// TIA Portal V20 export
FUNCTION "02 T5 EXCENTRIC HMI" : Void   // FC1218, LAD
TITLE = HMI
{ S7_Optimized_Access := 'TRUE' }
// stored: AutoNumber false, SetENOAutomatically false
BEGIN

REGION Network 1: Reset command interface from HMI in case of time-out
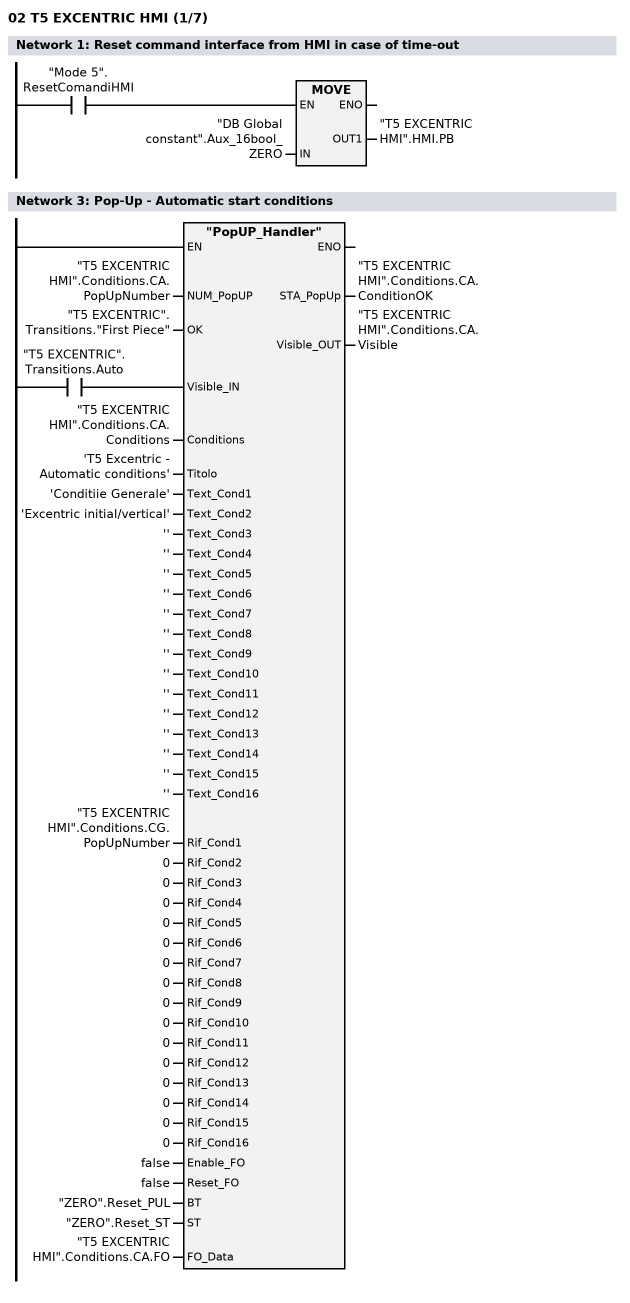
   RUNG wire#powerrail
      Contact( "Mode 5".ResetComandiHMI )
      Move(in := "DB Global constant".Aux_16bool_ZERO, out1 => "T5 EXCENTRIC HMI".HMI.PB)
   END_RUNG
   // the same network as SCL:
   IF "Mode 5".ResetComandiHMI THEN
       "T5 EXCENTRIC HMI".HMI.PB := "DB Global constant".Aux_16bool_ZERO;
   END_IF;
END_REGION

REGION Network 2: ============ POP UP ============
END_REGION

REGION Network 3: Pop-Up - Automatic start conditions
   RUNG wire#powerrail
      "PopUP_Handler"(Visible_IN := wire#w1, NUM_PopUP := "T5 EXCENTRIC HMI".Conditions.CA.PopUpNumber, OK := "T5 EXCENTRIC".Transitions."First Piece", Conditions := "T5 EXCENTRIC HMI".Conditions.CA.Conditions, Titolo := 'T5 Excentric - Automatic conditions', Text_Cond1 := 'Conditiie Generale', Text_Cond2 := 'Excentric initial/vertical', Text_Cond3 := '', Text_Cond4 := '', Text_Cond5 := '', Text_Cond6 := '', Text_Cond7 := '', Text_Cond8 := '', Text_Cond9 := '', Text_Cond10 := '', Text_Cond11 := '', Text_Cond12 := '', Text_Cond13 := '', Text_Cond14 := '', Text_Cond15 := '', Text_Cond16 := '', Rif_Cond1 := "T5 EXCENTRIC HMI".Conditions.CG.PopUpNumber, Rif_Cond2 := 0, Rif_Cond3 := 0, Rif_Cond4 := 0, Rif_Cond5 := 0, Rif_Cond6 := 0, Rif_Cond7 := 0, Rif_Cond8 := 0, Rif_Cond9 := 0, Rif_Cond10 := 0, Rif_Cond11 := 0, Rif_Cond12 := 0, Rif_Cond13 := 0, Rif_Cond14 := 0, Rif_Cond15 := 0, Rif_Cond16 := 0, Enable_FO := false, Reset_FO := false, BT := "ZERO".Reset_PUL, ST := "ZERO".Reset_ST, FO_Data := "T5 EXCENTRIC HMI".Conditions.CA.FO, STA_PopUp => "T5 EXCENTRIC HMI".Conditions.CA.ConditionOK, Visible_OUT => "T5 EXCENTRIC HMI".Conditions.CA.Visible)
   END_RUNG
   RUNG wire#powerrail
      Contact( "T5 EXCENTRIC".Transitions.Auto )
   END_RUNG wire#w1
   // the same network as SCL:
   "PopUP_Handler"(NUM_PopUP := "T5 EXCENTRIC HMI".Conditions.CA.PopUpNumber,
                   OK := "T5 EXCENTRIC".Transitions."First Piece",
                   Visible_IN := "T5 EXCENTRIC".Transitions.Auto,
                   Conditions := "T5 EXCENTRIC HMI".Conditions.CA.Conditions,
                   Titolo := 'T5 Excentric - Automatic conditions',
                   Text_Cond1 := 'Conditiie Generale',
                   Text_Cond2 := 'Excentric initial/vertical',
                   Text_Cond3 := '',
                   Text_Cond4 := '',
                   Text_Cond5 := '',
                   Text_Cond6 := '',
                   Text_Cond7 := '',
                   Text_Cond8 := '',
                   Text_Cond9 := '',
                   Text_Cond10 := '',
                   Text_Cond11 := '',
                   Text_Cond12 := '',
                   Text_Cond13 := '',
                   Text_Cond14 := '',
                   Text_Cond15 := '',
                   Text_Cond16 := '',
                   Rif_Cond1 := "T5 EXCENTRIC HMI".Conditions.CG.PopUpNumber,
                   Rif_Cond2 := 0,
                   Rif_Cond3 := 0,
                   Rif_Cond4 := 0,
                   Rif_Cond5 := 0,
                   Rif_Cond6 := 0,
                   Rif_Cond7 := 0,
                   Rif_Cond8 := 0,
                   Rif_Cond9 := 0,
                   Rif_Cond10 := 0,
                   Rif_Cond11 := 0,
                   Rif_Cond12 := 0,
                   Rif_Cond13 := 0,
                   Rif_Cond14 := 0,
                   Rif_Cond15 := 0,
                   Rif_Cond16 := 0,
                   Enable_FO := false,
                   Reset_FO := false,
                   BT := "ZERO".Reset_PUL,
                   ST := "ZERO".Reset_ST,
                   FO_Data := "T5 EXCENTRIC HMI".Conditions.CA.FO,
                   STA_PopUp => "T5 EXCENTRIC HMI".Conditions.CA.ConditionOK,
                   Visible_OUT => "T5 EXCENTRIC HMI".Conditions.CA.Visible);
END_REGION

REGION Network 4: Pop-Up - General conditions
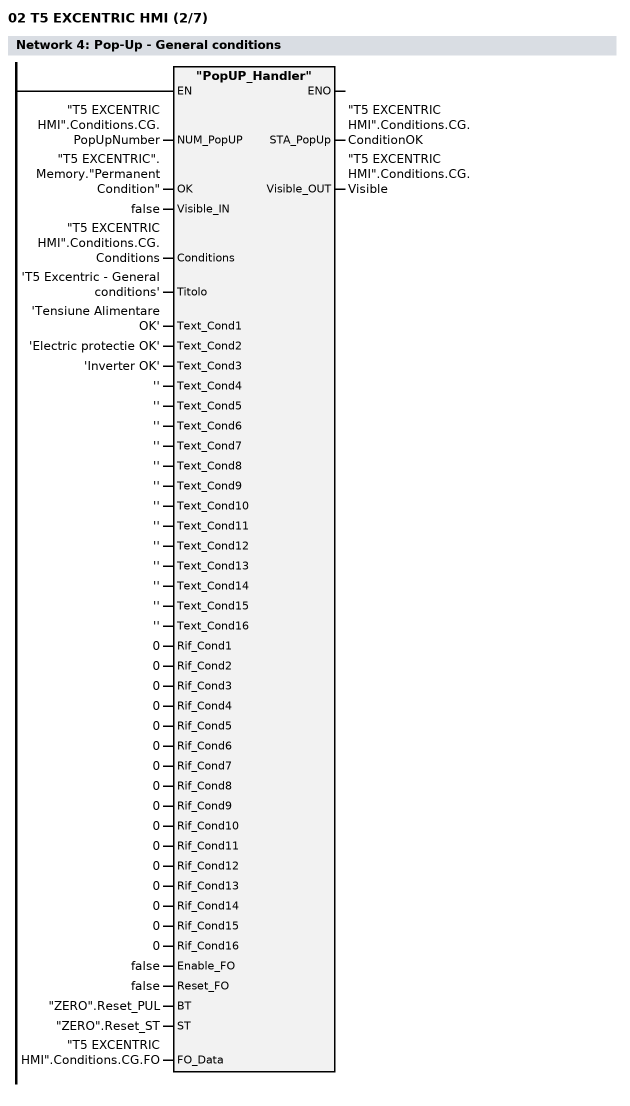
   RUNG wire#powerrail
      "PopUP_Handler"(NUM_PopUP := "T5 EXCENTRIC HMI".Conditions.CG.PopUpNumber, OK := "T5 EXCENTRIC".Memory."Permanent Condition", Visible_IN := false, Conditions := "T5 EXCENTRIC HMI".Conditions.CG.Conditions, Titolo := 'T5 Excentric - General conditions', Text_Cond1 := 'Tensiune Alimentare OK', Text_Cond2 := 'Electric protectie OK', Text_Cond3 := 'Inverter OK', Text_Cond4 := '', Text_Cond5 := '', Text_Cond6 := '', Text_Cond7 := '', Text_Cond8 := '', Text_Cond9 := '', Text_Cond10 := '', Text_Cond11 := '', Text_Cond12 := '', Text_Cond13 := '', Text_Cond14 := '', Text_Cond15 := '', Text_Cond16 := '', Rif_Cond1 := 0, Rif_Cond2 := 0, Rif_Cond3 := 0, Rif_Cond4 := 0, Rif_Cond5 := 0, Rif_Cond6 := 0, Rif_Cond7 := 0, Rif_Cond8 := 0, Rif_Cond9 := 0, Rif_Cond10 := 0, Rif_Cond11 := 0, Rif_Cond12 := 0, Rif_Cond13 := 0, Rif_Cond14 := 0, Rif_Cond15 := 0, Rif_Cond16 := 0, Enable_FO := false, Reset_FO := false, BT := "ZERO".Reset_PUL, ST := "ZERO".Reset_ST, FO_Data := "T5 EXCENTRIC HMI".Conditions.CG.FO, STA_PopUp => "T5 EXCENTRIC HMI".Conditions.CG.ConditionOK, Visible_OUT => "T5 EXCENTRIC HMI".Conditions.CG.Visible)
   END_RUNG
   // the same network as SCL:
   "PopUP_Handler"(NUM_PopUP := "T5 EXCENTRIC HMI".Conditions.CG.PopUpNumber,
                   OK := "T5 EXCENTRIC".Memory."Permanent Condition",
                   Visible_IN := false,
                   Conditions := "T5 EXCENTRIC HMI".Conditions.CG.Conditions,
                   Titolo := 'T5 Excentric - General conditions',
                   Text_Cond1 := 'Tensiune Alimentare OK',
                   Text_Cond2 := 'Electric protectie OK',
                   Text_Cond3 := 'Inverter OK',
                   Text_Cond4 := '',
                   Text_Cond5 := '',
                   Text_Cond6 := '',
                   Text_Cond7 := '',
                   Text_Cond8 := '',
                   Text_Cond9 := '',
                   Text_Cond10 := '',
                   Text_Cond11 := '',
                   Text_Cond12 := '',
                   Text_Cond13 := '',
                   Text_Cond14 := '',
                   Text_Cond15 := '',
                   Text_Cond16 := '',
                   Rif_Cond1 := 0,
                   Rif_Cond2 := 0,
                   Rif_Cond3 := 0,
                   Rif_Cond4 := 0,
                   Rif_Cond5 := 0,
                   Rif_Cond6 := 0,
                   Rif_Cond7 := 0,
                   Rif_Cond8 := 0,
                   Rif_Cond9 := 0,
                   Rif_Cond10 := 0,
                   Rif_Cond11 := 0,
                   Rif_Cond12 := 0,
                   Rif_Cond13 := 0,
                   Rif_Cond14 := 0,
                   Rif_Cond15 := 0,
                   Rif_Cond16 := 0,
                   Enable_FO := false,
                   Reset_FO := false,
                   BT := "ZERO".Reset_PUL,
                   ST := "ZERO".Reset_ST,
                   FO_Data := "T5 EXCENTRIC HMI".Conditions.CG.FO,
                   STA_PopUp => "T5 EXCENTRIC HMI".Conditions.CG.ConditionOK,
                   Visible_OUT => "T5 EXCENTRIC HMI".Conditions.CG.Visible);
END_REGION

REGION Network 5: Pop-Up - Cycle start conditions - Initial
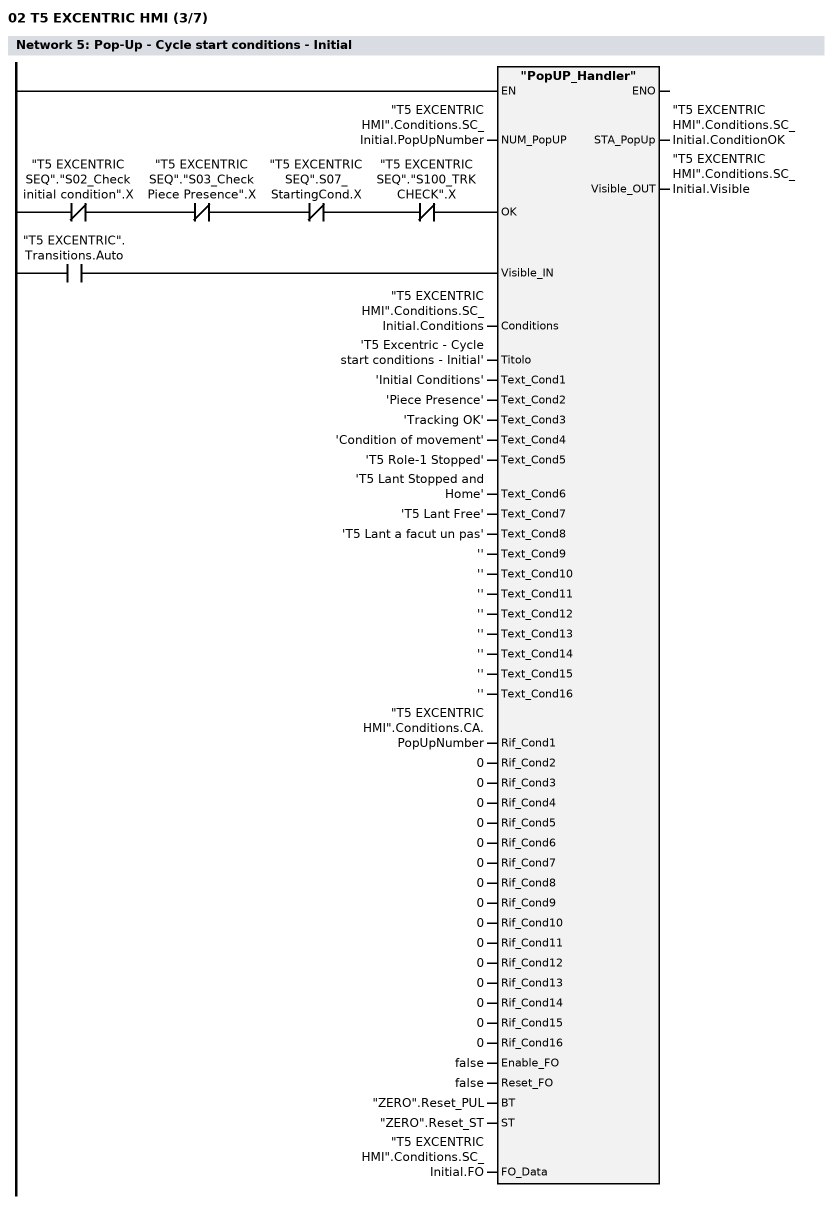
   RUNG wire#powerrail
      "PopUP_Handler"(OK := wire#w1, Visible_IN := wire#w2, NUM_PopUP := "T5 EXCENTRIC HMI".Conditions.SC_Initial.PopUpNumber, Conditions := "T5 EXCENTRIC HMI".Conditions.SC_Initial.Conditions, Titolo := 'T5 Excentric - Cycle start conditions - Initial', Text_Cond1 := 'Initial Conditions', Text_Cond2 := 'Piece Presence', Text_Cond3 := 'Tracking OK', Text_Cond4 := 'Condition of movement', Text_Cond5 := 'T5 Role-1 Stopped', Text_Cond6 := 'T5 Lant Stopped and Home', Text_Cond7 := 'T5 Lant Free', Text_Cond8 := 'T5 Lant a facut un pas', Text_Cond9 := '', Text_Cond10 := '', Text_Cond11 := '', Text_Cond12 := '', Text_Cond13 := '', Text_Cond14 := '', Text_Cond15 := '', Text_Cond16 := '', Rif_Cond1 := "T5 EXCENTRIC HMI".Conditions.CA.PopUpNumber, Rif_Cond2 := 0, Rif_Cond3 := 0, Rif_Cond4 := 0, Rif_Cond5 := 0, Rif_Cond6 := 0, Rif_Cond7 := 0, Rif_Cond8 := 0, Rif_Cond9 := 0, Rif_Cond10 := 0, Rif_Cond11 := 0, Rif_Cond12 := 0, Rif_Cond13 := 0, Rif_Cond14 := 0, Rif_Cond15 := 0, Rif_Cond16 := 0, Enable_FO := false, Reset_FO := false, BT := "ZERO".Reset_PUL, ST := "ZERO".Reset_ST, FO_Data := "T5 EXCENTRIC HMI".Conditions.SC_Initial.FO, STA_PopUp => "T5 EXCENTRIC HMI".Conditions.SC_Initial.ConditionOK, Visible_OUT => "T5 EXCENTRIC HMI".Conditions.SC_Initial.Visible)
   END_RUNG
   RUNG wire#powerrail
      I_Contact( "T5 EXCENTRIC SEQ"."S02_Check initial condition".X )
      I_Contact( "T5 EXCENTRIC SEQ"."S03_Check Piece Presence".X )
      I_Contact( "T5 EXCENTRIC SEQ".S07_StartingCond.X )
      I_Contact( "T5 EXCENTRIC SEQ"."S100_TRK CHECK".X )
   END_RUNG wire#w1
   RUNG wire#powerrail
      Contact( "T5 EXCENTRIC".Transitions.Auto )
   END_RUNG wire#w2
   // the same network as SCL:
   "PopUP_Handler"(NUM_PopUP := "T5 EXCENTRIC HMI".Conditions.SC_Initial.PopUpNumber,
                   OK := NOT "T5 EXCENTRIC SEQ"."S02_Check initial condition".X AND NOT "T5 EXCENTRIC SEQ"."S03_Check Piece Presence".X AND NOT "T5 EXCENTRIC SEQ".S07_StartingCond.X AND NOT "T5 EXCENTRIC SEQ"."S100_TRK CHECK".X,
                   Visible_IN := "T5 EXCENTRIC".Transitions.Auto,
                   Conditions := "T5 EXCENTRIC HMI".Conditions.SC_Initial.Conditions,
                   Titolo := 'T5 Excentric - Cycle start conditions - Initial',
                   Text_Cond1 := 'Initial Conditions',
                   Text_Cond2 := 'Piece Presence',
                   Text_Cond3 := 'Tracking OK',
                   Text_Cond4 := 'Condition of movement',
                   Text_Cond5 := 'T5 Role-1 Stopped',
                   Text_Cond6 := 'T5 Lant Stopped and Home',
                   Text_Cond7 := 'T5 Lant Free',
                   Text_Cond8 := 'T5 Lant a facut un pas',
                   Text_Cond9 := '',
                   Text_Cond10 := '',
                   Text_Cond11 := '',
                   Text_Cond12 := '',
                   Text_Cond13 := '',
                   Text_Cond14 := '',
                   Text_Cond15 := '',
                   Text_Cond16 := '',
                   Rif_Cond1 := "T5 EXCENTRIC HMI".Conditions.CA.PopUpNumber,
                   Rif_Cond2 := 0,
                   Rif_Cond3 := 0,
                   Rif_Cond4 := 0,
                   Rif_Cond5 := 0,
                   Rif_Cond6 := 0,
                   Rif_Cond7 := 0,
                   Rif_Cond8 := 0,
                   Rif_Cond9 := 0,
                   Rif_Cond10 := 0,
                   Rif_Cond11 := 0,
                   Rif_Cond12 := 0,
                   Rif_Cond13 := 0,
                   Rif_Cond14 := 0,
                   Rif_Cond15 := 0,
                   Rif_Cond16 := 0,
                   Enable_FO := false,
                   Reset_FO := false,
                   BT := "ZERO".Reset_PUL,
                   ST := "ZERO".Reset_ST,
                   FO_Data := "T5 EXCENTRIC HMI".Conditions.SC_Initial.FO,
                   STA_PopUp => "T5 EXCENTRIC HMI".Conditions.SC_Initial.ConditionOK,
                   Visible_OUT => "T5 EXCENTRIC HMI".Conditions.SC_Initial.Visible);
END_REGION

REGION Network 6: Pop-Up - Cycle start conditions - Vertical
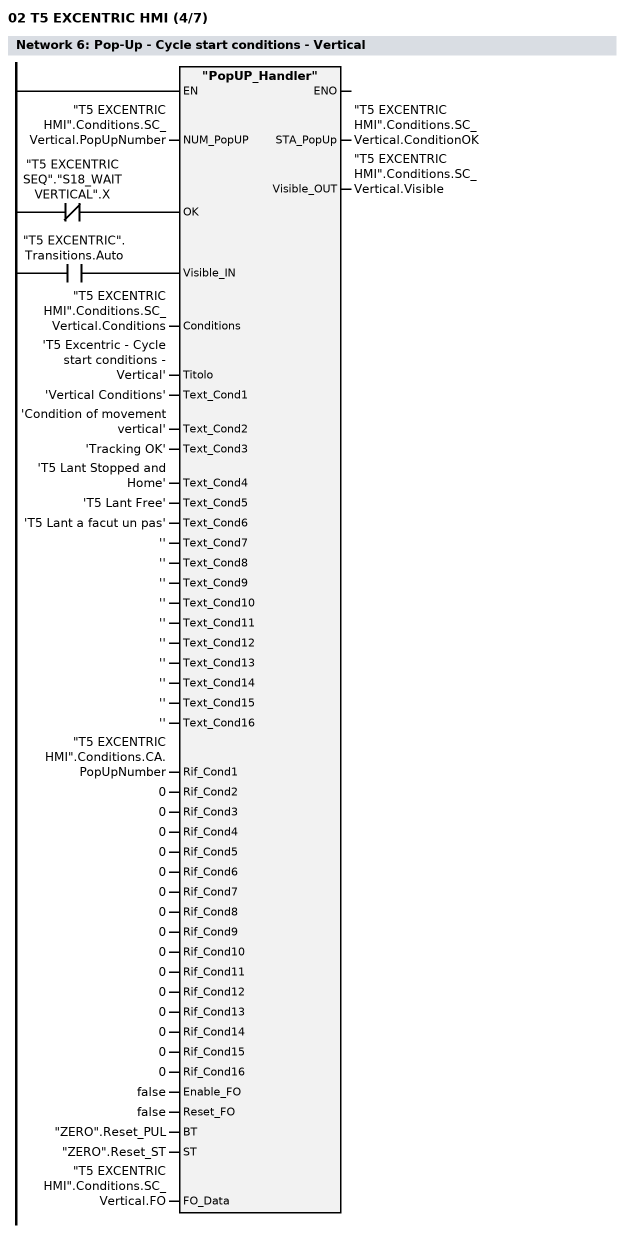
   RUNG wire#powerrail
      "PopUP_Handler"(OK := wire#w1, Visible_IN := wire#w2, NUM_PopUP := "T5 EXCENTRIC HMI".Conditions.SC_Vertical.PopUpNumber, Conditions := "T5 EXCENTRIC HMI".Conditions.SC_Vertical.Conditions, Titolo := 'T5 Excentric - Cycle start conditions - Vertical', Text_Cond1 := 'Vertical Conditions', Text_Cond2 := 'Condition of movement vertical', Text_Cond3 := 'Tracking OK', Text_Cond4 := 'T5 Lant Stopped and Home', Text_Cond5 := 'T5 Lant Free', Text_Cond6 := 'T5 Lant a facut un pas', Text_Cond7 := '', Text_Cond8 := '', Text_Cond9 := '', Text_Cond10 := '', Text_Cond11 := '', Text_Cond12 := '', Text_Cond13 := '', Text_Cond14 := '', Text_Cond15 := '', Text_Cond16 := '', Rif_Cond1 := "T5 EXCENTRIC HMI".Conditions.CA.PopUpNumber, Rif_Cond2 := 0, Rif_Cond3 := 0, Rif_Cond4 := 0, Rif_Cond5 := 0, Rif_Cond6 := 0, Rif_Cond7 := 0, Rif_Cond8 := 0, Rif_Cond9 := 0, Rif_Cond10 := 0, Rif_Cond11 := 0, Rif_Cond12 := 0, Rif_Cond13 := 0, Rif_Cond14 := 0, Rif_Cond15 := 0, Rif_Cond16 := 0, Enable_FO := false, Reset_FO := false, BT := "ZERO".Reset_PUL, ST := "ZERO".Reset_ST, FO_Data := "T5 EXCENTRIC HMI".Conditions.SC_Vertical.FO, STA_PopUp => "T5 EXCENTRIC HMI".Conditions.SC_Vertical.ConditionOK, Visible_OUT => "T5 EXCENTRIC HMI".Conditions.SC_Vertical.Visible)
   END_RUNG
   RUNG wire#powerrail
      I_Contact( "T5 EXCENTRIC SEQ"."S18_WAIT VERTICAL".X )
   END_RUNG wire#w1
   RUNG wire#powerrail
      Contact( "T5 EXCENTRIC".Transitions.Auto )
   END_RUNG wire#w2
   // the same network as SCL:
   "PopUP_Handler"(NUM_PopUP := "T5 EXCENTRIC HMI".Conditions.SC_Vertical.PopUpNumber,
                   OK := NOT "T5 EXCENTRIC SEQ"."S18_WAIT VERTICAL".X,
                   Visible_IN := "T5 EXCENTRIC".Transitions.Auto,
                   Conditions := "T5 EXCENTRIC HMI".Conditions.SC_Vertical.Conditions,
                   Titolo := 'T5 Excentric - Cycle start conditions - Vertical',
                   Text_Cond1 := 'Vertical Conditions',
                   Text_Cond2 := 'Condition of movement vertical',
                   Text_Cond3 := 'Tracking OK',
                   Text_Cond4 := 'T5 Lant Stopped and Home',
                   Text_Cond5 := 'T5 Lant Free',
                   Text_Cond6 := 'T5 Lant a facut un pas',
                   Text_Cond7 := '',
                   Text_Cond8 := '',
                   Text_Cond9 := '',
                   Text_Cond10 := '',
                   Text_Cond11 := '',
                   Text_Cond12 := '',
                   Text_Cond13 := '',
                   Text_Cond14 := '',
                   Text_Cond15 := '',
                   Text_Cond16 := '',
                   Rif_Cond1 := "T5 EXCENTRIC HMI".Conditions.CA.PopUpNumber,
                   Rif_Cond2 := 0,
                   Rif_Cond3 := 0,
                   Rif_Cond4 := 0,
                   Rif_Cond5 := 0,
                   Rif_Cond6 := 0,
                   Rif_Cond7 := 0,
                   Rif_Cond8 := 0,
                   Rif_Cond9 := 0,
                   Rif_Cond10 := 0,
                   Rif_Cond11 := 0,
                   Rif_Cond12 := 0,
                   Rif_Cond13 := 0,
                   Rif_Cond14 := 0,
                   Rif_Cond15 := 0,
                   Rif_Cond16 := 0,
                   Enable_FO := false,
                   Reset_FO := false,
                   BT := "ZERO".Reset_PUL,
                   ST := "ZERO".Reset_ST,
                   FO_Data := "T5 EXCENTRIC HMI".Conditions.SC_Vertical.FO,
                   STA_PopUp => "T5 EXCENTRIC HMI".Conditions.SC_Vertical.ConditionOK,
                   Visible_OUT => "T5 EXCENTRIC HMI".Conditions.SC_Vertical.Visible);
END_REGION

REGION Network 7: Pop-Up - Conditions of movement FORWARD
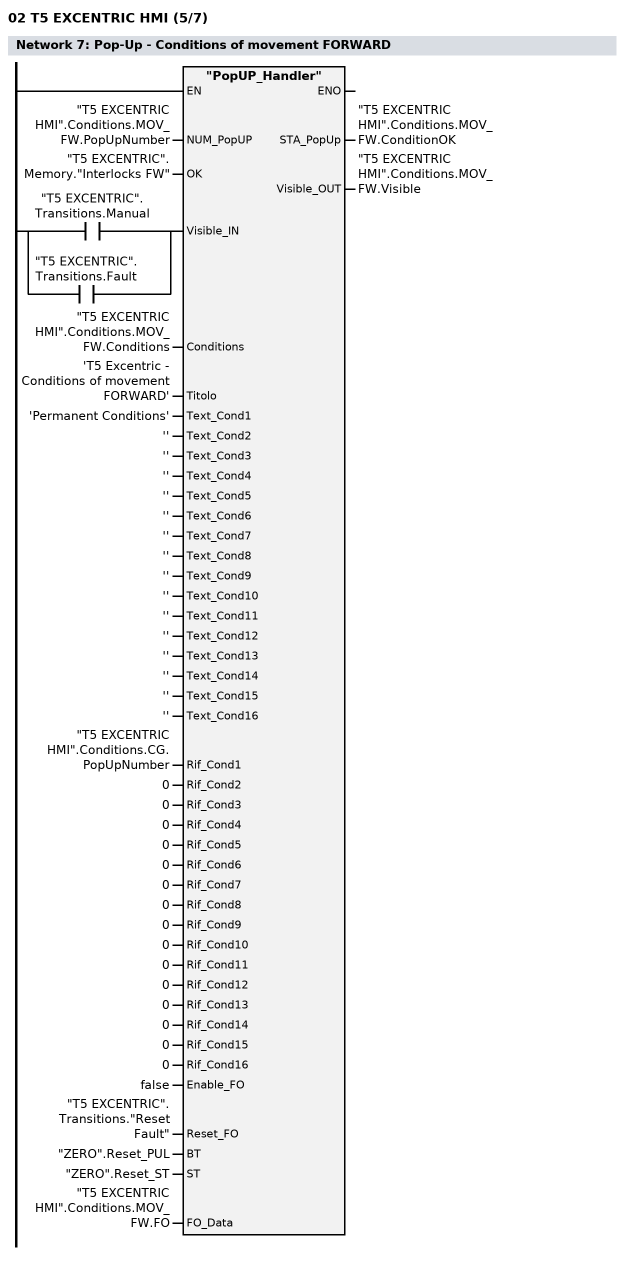
   RUNG wire#powerrail
      "PopUP_Handler"(Visible_IN := wire#w1, NUM_PopUP := "T5 EXCENTRIC HMI".Conditions.MOV_FW.PopUpNumber, OK := "T5 EXCENTRIC".Memory."Interlocks FW", Conditions := "T5 EXCENTRIC HMI".Conditions.MOV_FW.Conditions, Titolo := 'T5 Excentric - Conditions of movement FORWARD', Text_Cond1 := 'Permanent Conditions', Text_Cond2 := '', Text_Cond3 := '', Text_Cond4 := '', Text_Cond5 := '', Text_Cond6 := '', Text_Cond7 := '', Text_Cond8 := '', Text_Cond9 := '', Text_Cond10 := '', Text_Cond11 := '', Text_Cond12 := '', Text_Cond13 := '', Text_Cond14 := '', Text_Cond15 := '', Text_Cond16 := '', Rif_Cond1 := "T5 EXCENTRIC HMI".Conditions.CG.PopUpNumber, Rif_Cond2 := 0, Rif_Cond3 := 0, Rif_Cond4 := 0, Rif_Cond5 := 0, Rif_Cond6 := 0, Rif_Cond7 := 0, Rif_Cond8 := 0, Rif_Cond9 := 0, Rif_Cond10 := 0, Rif_Cond11 := 0, Rif_Cond12 := 0, Rif_Cond13 := 0, Rif_Cond14 := 0, Rif_Cond15 := 0, Rif_Cond16 := 0, Enable_FO := false, Reset_FO := "T5 EXCENTRIC".Transitions."Reset Fault", BT := "ZERO".Reset_PUL, ST := "ZERO".Reset_ST, FO_Data := "T5 EXCENTRIC HMI".Conditions.MOV_FW.FO, STA_PopUp => "T5 EXCENTRIC HMI".Conditions.MOV_FW.ConditionOK, Visible_OUT => "T5 EXCENTRIC HMI".Conditions.MOV_FW.Visible)
   END_RUNG
   RUNG wire#powerrail
      Contact( "T5 EXCENTRIC".Transitions.Manual )
   END_RUNG wire#w1
   RUNG wire#powerrail
      Contact( "T5 EXCENTRIC".Transitions.Fault )
   END_RUNG wire#w1
   // the same network as SCL:
   "PopUP_Handler"(NUM_PopUP := "T5 EXCENTRIC HMI".Conditions.MOV_FW.PopUpNumber,
                   OK := "T5 EXCENTRIC".Memory."Interlocks FW",
                   Visible_IN := "T5 EXCENTRIC".Transitions.Manual OR "T5 EXCENTRIC".Transitions.Fault,
                   Conditions := "T5 EXCENTRIC HMI".Conditions.MOV_FW.Conditions,
                   Titolo := 'T5 Excentric - Conditions of movement FORWARD',
                   Text_Cond1 := 'Permanent Conditions',
                   Text_Cond2 := '',
                   Text_Cond3 := '',
                   Text_Cond4 := '',
                   Text_Cond5 := '',
                   Text_Cond6 := '',
                   Text_Cond7 := '',
                   Text_Cond8 := '',
                   Text_Cond9 := '',
                   Text_Cond10 := '',
                   Text_Cond11 := '',
                   Text_Cond12 := '',
                   Text_Cond13 := '',
                   Text_Cond14 := '',
                   Text_Cond15 := '',
                   Text_Cond16 := '',
                   Rif_Cond1 := "T5 EXCENTRIC HMI".Conditions.CG.PopUpNumber,
                   Rif_Cond2 := 0,
                   Rif_Cond3 := 0,
                   Rif_Cond4 := 0,
                   Rif_Cond5 := 0,
                   Rif_Cond6 := 0,
                   Rif_Cond7 := 0,
                   Rif_Cond8 := 0,
                   Rif_Cond9 := 0,
                   Rif_Cond10 := 0,
                   Rif_Cond11 := 0,
                   Rif_Cond12 := 0,
                   Rif_Cond13 := 0,
                   Rif_Cond14 := 0,
                   Rif_Cond15 := 0,
                   Rif_Cond16 := 0,
                   Enable_FO := false,
                   Reset_FO := "T5 EXCENTRIC".Transitions."Reset Fault",
                   BT := "ZERO".Reset_PUL,
                   ST := "ZERO".Reset_ST,
                   FO_Data := "T5 EXCENTRIC HMI".Conditions.MOV_FW.FO,
                   STA_PopUp => "T5 EXCENTRIC HMI".Conditions.MOV_FW.ConditionOK,
                   Visible_OUT => "T5 EXCENTRIC HMI".Conditions.MOV_FW.Visible);
END_REGION

REGION Network 8: Pop-Up - Conditions of movement BACKWARD
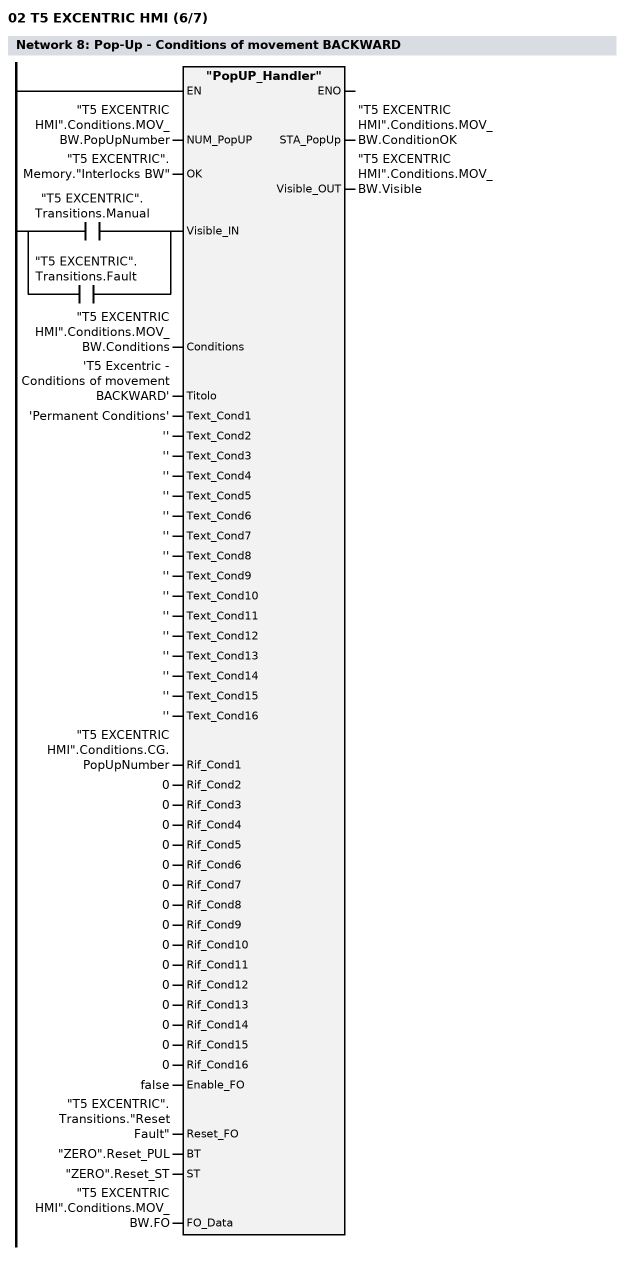
   RUNG wire#powerrail
      "PopUP_Handler"(Visible_IN := wire#w1, NUM_PopUP := "T5 EXCENTRIC HMI".Conditions.MOV_BW.PopUpNumber, OK := "T5 EXCENTRIC".Memory."Interlocks BW", Conditions := "T5 EXCENTRIC HMI".Conditions.MOV_BW.Conditions, Titolo := 'T5 Excentric - Conditions of movement BACKWARD', Text_Cond1 := 'Permanent Conditions', Text_Cond2 := '', Text_Cond3 := '', Text_Cond4 := '', Text_Cond5 := '', Text_Cond6 := '', Text_Cond7 := '', Text_Cond8 := '', Text_Cond9 := '', Text_Cond10 := '', Text_Cond11 := '', Text_Cond12 := '', Text_Cond13 := '', Text_Cond14 := '', Text_Cond15 := '', Text_Cond16 := '', Rif_Cond1 := "T5 EXCENTRIC HMI".Conditions.CG.PopUpNumber, Rif_Cond2 := 0, Rif_Cond3 := 0, Rif_Cond4 := 0, Rif_Cond5 := 0, Rif_Cond6 := 0, Rif_Cond7 := 0, Rif_Cond8 := 0, Rif_Cond9 := 0, Rif_Cond10 := 0, Rif_Cond11 := 0, Rif_Cond12 := 0, Rif_Cond13 := 0, Rif_Cond14 := 0, Rif_Cond15 := 0, Rif_Cond16 := 0, Enable_FO := false, Reset_FO := "T5 EXCENTRIC".Transitions."Reset Fault", BT := "ZERO".Reset_PUL, ST := "ZERO".Reset_ST, FO_Data := "T5 EXCENTRIC HMI".Conditions.MOV_BW.FO, STA_PopUp => "T5 EXCENTRIC HMI".Conditions.MOV_BW.ConditionOK, Visible_OUT => "T5 EXCENTRIC HMI".Conditions.MOV_BW.Visible)
   END_RUNG
   RUNG wire#powerrail
      Contact( "T5 EXCENTRIC".Transitions.Manual )
   END_RUNG wire#w1
   RUNG wire#powerrail
      Contact( "T5 EXCENTRIC".Transitions.Fault )
   END_RUNG wire#w1
   // the same network as SCL:
   "PopUP_Handler"(NUM_PopUP := "T5 EXCENTRIC HMI".Conditions.MOV_BW.PopUpNumber,
                   OK := "T5 EXCENTRIC".Memory."Interlocks BW",
                   Visible_IN := "T5 EXCENTRIC".Transitions.Manual OR "T5 EXCENTRIC".Transitions.Fault,
                   Conditions := "T5 EXCENTRIC HMI".Conditions.MOV_BW.Conditions,
                   Titolo := 'T5 Excentric - Conditions of movement BACKWARD',
                   Text_Cond1 := 'Permanent Conditions',
                   Text_Cond2 := '',
                   Text_Cond3 := '',
                   Text_Cond4 := '',
                   Text_Cond5 := '',
                   Text_Cond6 := '',
                   Text_Cond7 := '',
                   Text_Cond8 := '',
                   Text_Cond9 := '',
                   Text_Cond10 := '',
                   Text_Cond11 := '',
                   Text_Cond12 := '',
                   Text_Cond13 := '',
                   Text_Cond14 := '',
                   Text_Cond15 := '',
                   Text_Cond16 := '',
                   Rif_Cond1 := "T5 EXCENTRIC HMI".Conditions.CG.PopUpNumber,
                   Rif_Cond2 := 0,
                   Rif_Cond3 := 0,
                   Rif_Cond4 := 0,
                   Rif_Cond5 := 0,
                   Rif_Cond6 := 0,
                   Rif_Cond7 := 0,
                   Rif_Cond8 := 0,
                   Rif_Cond9 := 0,
                   Rif_Cond10 := 0,
                   Rif_Cond11 := 0,
                   Rif_Cond12 := 0,
                   Rif_Cond13 := 0,
                   Rif_Cond14 := 0,
                   Rif_Cond15 := 0,
                   Rif_Cond16 := 0,
                   Enable_FO := false,
                   Reset_FO := "T5 EXCENTRIC".Transitions."Reset Fault",
                   BT := "ZERO".Reset_PUL,
                   ST := "ZERO".Reset_ST,
                   FO_Data := "T5 EXCENTRIC HMI".Conditions.MOV_BW.FO,
                   STA_PopUp => "T5 EXCENTRIC HMI".Conditions.MOV_BW.ConditionOK,
                   Visible_OUT => "T5 EXCENTRIC HMI".Conditions.MOV_BW.Visible);
END_REGION

REGION Network 9: ============ HMI STATE ============
END_REGION

REGION Network 10: HMI Status - Commands
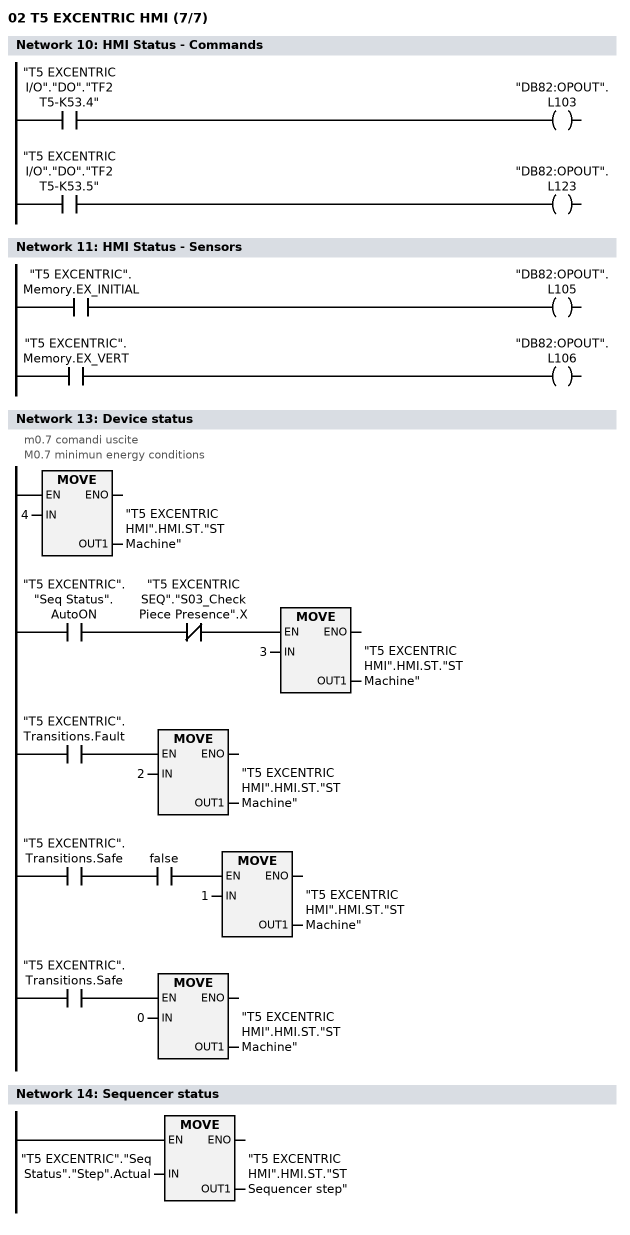
   RUNG wire#powerrail
      Contact( "T5 EXCENTRIC I/O"."DO"."TF2 T5-K53.4" )
      Coil( "DB82:OPOUT".L103 )
   END_RUNG
   RUNG wire#powerrail
      Contact( "T5 EXCENTRIC I/O"."DO"."TF2 T5-K53.5" )
      Coil( "DB82:OPOUT".L123 )
   END_RUNG
   // the same network as SCL:
   "DB82:OPOUT".L103 := "T5 EXCENTRIC I/O"."DO"."TF2 T5-K53.4";
   "DB82:OPOUT".L123 := "T5 EXCENTRIC I/O"."DO"."TF2 T5-K53.5";
END_REGION

REGION Network 11: HMI Status - Sensors
   RUNG wire#powerrail
      Contact( "T5 EXCENTRIC".Memory.EX_INITIAL )
      Coil( "DB82:OPOUT".L105 )
   END_RUNG
   RUNG wire#powerrail
      Contact( "T5 EXCENTRIC".Memory.EX_VERT )
      Coil( "DB82:OPOUT".L106 )
   END_RUNG
   // the same network as SCL:
   "DB82:OPOUT".L105 := "T5 EXCENTRIC".Memory.EX_INITIAL;
   "DB82:OPOUT".L106 := "T5 EXCENTRIC".Memory.EX_VERT;
END_REGION

REGION Network 12: HMI Status - Alarma
END_REGION

REGION Network 13: Device status
   // m0.7 comandi uscite
   // M0.7 minimun energy conditions
   RUNG wire#powerrail
      Move(in := 4, out1 => "T5 EXCENTRIC HMI".HMI.ST."ST Machine")
   END_RUNG
   RUNG wire#powerrail
      Contact( "T5 EXCENTRIC"."Seq Status".AutoON )
      I_Contact( "T5 EXCENTRIC SEQ"."S03_Check Piece Presence".X )
      Move(in := 3, out1 => "T5 EXCENTRIC HMI".HMI.ST."ST Machine")
   END_RUNG
   RUNG wire#powerrail
      Contact( "T5 EXCENTRIC".Transitions.Fault )
      Move(in := 2, out1 => "T5 EXCENTRIC HMI".HMI.ST."ST Machine")
   END_RUNG
   RUNG wire#powerrail
      Contact( "T5 EXCENTRIC".Transitions.Safe )
      Contact( false )
      Move(in := 1, out1 => "T5 EXCENTRIC HMI".HMI.ST."ST Machine")
   END_RUNG
   RUNG wire#powerrail
      Contact( "T5 EXCENTRIC".Transitions.Safe )
      Move(in := 0, out1 => "T5 EXCENTRIC HMI".HMI.ST."ST Machine")
   END_RUNG
   // the same network as SCL:
   "T5 EXCENTRIC HMI".HMI.ST."ST Machine" := 4;
   IF "T5 EXCENTRIC"."Seq Status".AutoON AND NOT "T5 EXCENTRIC SEQ"."S03_Check Piece Presence".X THEN
       "T5 EXCENTRIC HMI".HMI.ST."ST Machine" := 3;
   END_IF;
   IF "T5 EXCENTRIC".Transitions.Fault THEN "T5 EXCENTRIC HMI".HMI.ST."ST Machine" := 2; END_IF;
   IF "T5 EXCENTRIC".Transitions.Safe AND false THEN "T5 EXCENTRIC HMI".HMI.ST."ST Machine" := 1; END_IF;
   IF "T5 EXCENTRIC".Transitions.Safe THEN "T5 EXCENTRIC HMI".HMI.ST."ST Machine" := 0; END_IF;
END_REGION

REGION Network 14: Sequencer status
   RUNG wire#powerrail
      Move(in := "T5 EXCENTRIC"."Seq Status"."Step".Actual, out1 => "T5 EXCENTRIC HMI".HMI.ST."ST Sequencer step")
   END_RUNG
   // the same network as SCL:
   "T5 EXCENTRIC HMI".HMI.ST."ST Sequencer step" := "T5 EXCENTRIC"."Seq Status"."Step".Actual;
END_REGION
END_FUNCTION
